FUNCTION_BLOCK Motor_Inversor_Automatico_Unico (* Composite Function Block Type *)
  (* Standard: 61499-2 *)
  (* Version 0.0, 1/22/2026, Schneider Electric, template *)
  PACKAGE Hidryco.HidrycoLib;
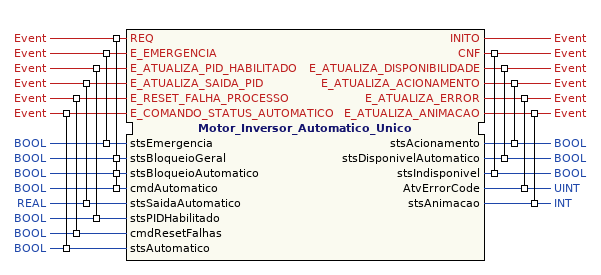
  EVENT_INPUT
    REQ WITH stsBloqueioGeral, stsBloqueioAutomatico, cmdAutomatico; (* Normal Execution Request *)
    E_EMERGENCIA WITH stsEmergencia;
    E_ATUALIZA_PID_HABILITADO WITH stsPIDHabilitado;
    E_ATUALIZA_SAIDA_PID WITH stsSaidaAutomatico;
    E_RESET_FALHA_PROCESSO WITH cmdResetFalhas;
    E_COMANDO_STATUS_AUTOMATICO WITH stsAutomatico;
  END_EVENT
  EVENT_OUTPUT
    INITO; (* Initialization Confirm *)
    CNF WITH stsIndisponivel; (* Execution Confirmation *)
    E_ATUALIZA_DISPONIBILIDADE WITH stsDisponivelAutomatico;
    E_ATUALIZA_ACIONAMENTO WITH stsAcionamento;
    E_ATUALIZA_ERROR WITH AtvErrorCode;
    E_ATUALIZA_ANIMACAO WITH stsAnimacao;
  END_EVENT
  VAR_INPUT
    stsEmergencia : BOOL;
    stsBloqueioGeral : BOOL;
    stsBloqueioAutomatico : BOOL;
    cmdAutomatico : BOOL;
    stsSaidaAutomatico : REAL;
    stsPIDHabilitado : BOOL;
    cmdResetFalhas : BOOL;
    stsAutomatico : BOOL; (* Botão unico que deixa em automatico *)
  END_VAR
  VAR_OUTPUT
    stsAcionamento : BOOL;
    stsDisponivelAutomatico : BOOL;
    stsIndisponivel : BOOL;
    AtvErrorCode : UINT; (* Current value(i) in the named variable array element *)
    stsAnimacao : INT;
  END_VAR
  (* 0 - INITIALIZATION *)
  (* 1 - FUNCTIONAL INPUT INTERFACE *)
  (* 6 - OT-IT INTERFACE *)
  (* 2 - FUNCTIONAL OUTPUT INTERFACE *)
  (* 3 - FIELD INTERFACE *)
  (* 4 - CHILDREN *)
  (* 5 - LOGICS *)
  (* 5.B - OPERATION MODE MANAGEMENT *)
  (* 5.D - INTERLOCKS MANAGEMENT *)
  (* 5.A - FUNCTIONAL BEHAVIORS *)
  (* 5.C - INTERLOCKS MANAGEMENT *)
  FBS
    IThis : Motor_Inversor_Automatico_Unico_HMI(QI := TRUE);
    SYMLINKMULTIVARDST1 : SYMLINKMULTIVARDST_151ACB50A2F8223B2(QI := TRUE, NAME1 := '$${PATH}stsFalhaComunicacao', NAME2 := '$${PATH}stsRemoto', NAME3 := '$${PATH}stsLocal'); {SET_ATTRIBUTE(Configuration.GenericFBType.InterfaceParams, Runtime.System#I:=3;VALUE${I$}:BOOL,BOOL,BOOL)}
    Inversor : ATV_Schneider;
    plcStart1 : plcStart(Prio := 5);
  END_FBS
  EVENT_CONNECTIONS
    E_EMERGENCIA TO Inversor.E_QUICK_STOP;
    Inversor.E_ERROR TO E_ATUALIZA_ERROR;
    E_RESET_FALHA_PROCESSO TO Inversor.E_RESET;
    SYMLINKMULTIVARDST1.INITO TO plcStart1.ACK_FIRST;
    plcStart1.FIRST_INIT TO IThis.77A2F60CB33ACCE3;
    plcStart1.REDO_INIT TO IThis.77A2F60CB33ACCE3;
    REQ TO IThis.3E1D0BBAE7B97111;
    Inversor.E_STATUS TO IThis.3E1D0BBAE7B97111;
    IThis.E95E96A346CBF4D4 TO IThis.8E9224D666F3049B;
    E_COMANDO_STATUS_AUTOMATICO TO IThis.8E9224D666F3049B;
    IThis.8988C31EE2188F23 TO SYMLINKMULTIVARDST1.INIT;
  END_CONNECTIONS
  DATA_CONNECTIONS
    stsEmergencia TO Inversor.CommandQuickStop;
    Inversor.AtvErrorCode TO AtvErrorCode;
    SYMLINKMULTIVARDST1.VALUE2 TO IThis.841BF87C17BC0349;
    stsAutomatico TO IThis.275D60C0FD2DF838;
    IThis.89F4F7CACE4761CD TO IThis.6EDA2309B49292B1;
    Inversor.stsVelocidade TO IThis.E981264F18CB1FBA;
    Inversor.stsCorrente TO IThis.A3116B301DAF6FAE;
    Inversor.stsFrequencia TO IThis.DBB52AC5CACB9985;
    Inversor.stsTensao TO IThis.EDC39F8AA815428B;
    Inversor.stsTorque TO IThis.395035782FFD9074;
    Inversor.stsPotencia TO IThis.4407C745574824E4;
  END_CONNECTIONS
END_FUNCTION_BLOCK
